// TIA Portal V19 export
VAR_GLOBAL   // PLC tag table "01_SAFETY_Q"
   FDo_C_CambioFormato_Bordatrice AT %Q1000.1 : Bool;   // 0DO1 - 169KA1/KA2
   FDo_C_HU_Pareggiatore_STO_CYTROPACK AT %Q1000.5 : Bool;   // 0DO5 - 280KA1/KA2
   FDo_C_HU_Aspo AT %Q1000.2 : Bool;   // 0DO2 - 206KA1/KA2 Motoe pompa C.Olio Aspi
   FDo_V_Air_A0301_A0302 AT %Q1558.0 : Bool;   // 200DO0 - 180YV1 - Valvola taglio aria A0301 (Ribaltamento) + A0302 ingresso (bordatrice)
   FDo_EStop_Coda_BloccaggioCremagliera_PistonePareggLong AT %Q1414.0 : Bool;   // 300DO0 - 284KA1/KA2
   FDo_V_Air_A0302_A0303 AT %Q1420.0 : Bool;   // 310DO0 - 182YV1 - Valvola taglio aria zona pareggiamento e preparazione pacco
   FDo_Ev_Stand_BY_HU_Pareggiatore AT %Q1420.1 : Bool;   // 310D01 - 282YV1
   FDo_EStop_Testa_BloccaggioCremagliera AT %Q1507.0 : Bool;   // 286KA1/KA2 - 350DO0
   FDo_C_HU_Area01 AT %Q1000.3 : Bool;   // 0DO3 - 220KA1/KA2 Motore pompa C.Olio Area 01
   FDo_C_HU_FinalCut AT %Q1000.4 : Bool;   // 0DO4 - 248KA1/KA2
   FDo_V_DecoilersHorizRot AT %Q1093.0 : Bool;   // 100DO0 - 206KA3/KA4
   FDo_V_Aspo_1 AT %Q1093.1 : Bool;   // 100DO1 - 206KA5/KA6 Contattore c/Feedback
   FDo_V_Aspo_2 AT %Q1093.2 : Bool;   // 100DO2 - 206KA7/KA8 Contattore c/Feedback
   FDo_V_CoilCar AT %Q1093.3 : Bool;   // 100DO3 - 222KA1/KA2
   FDo_V_Peeler AT %Q1093.4 : Bool;   // 100DO4 - 224KA1/KA2
   FDo_V_FinalCut AT %Q1093.5 : Bool;   // 100DO5 - 250KA1/KA2
   FDo_V_Air_Gen AT %Q1107.0 : Bool;   // 110DO0 - 174YV1
   FDo_V_StandBY_HU_Aspo AT %Q1107.1 : Bool;   // 110D01 - 208YV1
   FDo_V_StandBY_HU_Area01 AT %Q1107.2 : Bool;   // 110D02 - 221YV1
   FDo_V_Accumulatore_HU_Area01 AT %Q1107.3 : Bool;   // 110DO3 - 221YV2
   FDo_V_JB_Cut_Rest AT %Q1112.0 : Bool;   // 111DO0 - 226YV1
   FDo_V_JB_Cut_Work AT %Q1112.1 : Bool;   // 111DO1 - 226YV2
   FDo_V_StandBY_HU_FinalCut AT %Q1117.0 : Bool;   // 120DO0 - 249YV1
   FDo_V_Accumulatore_HU_FinalCut AT %Q1117.1 : Bool;   // 120DO1 - 249YV2
   FDo_C_CambioFormato_Profilatrice AT %Q1000.0 : Bool;   // 0DO0 - 168KA1/KA2
   Fdbk_V_DecoilersHorizRot_Ch1 AT %I104.6 : Bool;   // 209SQ1
   Fdbk_V_DecoilersHorizRot_Ch2 AT %I104.7 : Bool;   // 209SQ1
   Fdbk_V_Aspo01_Ch1 AT %I105.0 : Bool;   // 210SQ1
   Fdbk_V_Aspo01_Ch2 AT %I105.1 : Bool;   // 210SQ1
   Fdbk_V_Aspo02_Ch1 AT %I105.2 : Bool;   // 212SQ1
   Fdbk_V_Aspo02_Ch2 AT %I105.3 : Bool;   // 212SQ1
   Fbdk_V_CoilCar_Ch1 AT %I105.4 : Bool;   // 222SQ1
   Fbdk_V_CoilCar_Ch2 AT %I105.5 : Bool;   // 222SQ1
   Fbdk_V_Peeler_Ch1 AT %I105.6 : Bool;   // 224SQ1
   Fbdk_V_Peeler_Ch2 AT %I105.7 : Bool;   // 224SQ1
   Fbdk_V_JB_Cut_Ch1 AT %I106.0 : Bool;   // 226SQ1
   Fdbk_V_FinalCut_Ch1 AT %I108.6 : Bool;   // 250SQ1
   Fdbk_V_FinalCut_Ch2 AT %I108.7 : Bool;   // 250SQ1
   Fdbk_V_Air_Gen_Ch1 AT %I102.4 : Bool;   // 174SQ1
   Fdbk_V_Air_Gen_Ch2 AT %I102.3 : Bool;   // 174SQ1
   Fdbk_FDo_Bloccaggio_Valve AT %I360.1 : Bool;   // 286KA1/KA2
   Fbkk_C_Sezionatrice_FinalCut AT %I101.5 : Bool;   // 250KA1/KA2
   Fdbk_C_Peeler AT %I101.3 : Bool;   // 224KA1/KA2
   Fdbk_C_CoilCar AT %I101.2 : Bool;   // 222KA1/KA2
   "HU_B.Taglio_Motore_Controllo_Sicurezza" AT %I6.5 : Bool;   // 248KA1/KA2
   Fdbk_FDo_Bloccaggio_Pareggiatore_Valves AT %I309.5 : Bool;   // 284KA1
   FDo_V_Air_A0304 AT %Q1420.2 : Bool;   // 310DO2 - 183YV1
   FDo_EStop_Coda_BloccaggioCremagliera_PistonePareggLong_VS AT %I1414.0 : Bool;   // 300DO0 - 284KA1/KA2
   FDo_EStop_Testa_BloccaggioCremagliera_VS AT %I1507.0 : Bool;   // 286KA1/KA2 - 350DO0
   QBAD_FDo_C_CambioFormato_Bordatrice AT %I1000.1 : Bool;
   QBAD_FDo_C_CambioFormato_Profilatrice AT %I1000.0 : Bool;
   QBAD_FDo_C_HU_Aspo AT %I1000.2 : Bool;
   QBAD_FDo_C_HU_Area01 AT %I1000.3 : Bool;
   QBAD_FDo_C_HU_FinalCut AT %I1000.4 : Bool;
   QBAD_FDo_FDo_C_HU_Pareggiatore_STO_CYTROPACK AT %I1000.5 : Bool;
   QBAD_FDo_V_DecoilersHorizRot AT %I1093.0 : Bool;
   QBAD_FDo_V_Aspo_1 AT %I1093.1 : Bool;
   QBAD_FDo_V_Aspo_2 AT %I1093.2 : Bool;
   QBAD_FDo_V_CoilCar AT %I1093.3 : Bool;
   QBAD_FDo_V_Peeler AT %I1093.4 : Bool;
   QBAD_FDo_V_JB_Cut_Rest AT %I1112.0 : Bool;
   QBAD_FDo_V_JB_Cut_Work AT %I1112.1 : Bool;
   Fdbk_C_Aspo01 AT %I101.0 : Bool;   // 206KA5 / KA6
   Fdbk_C_Aspo02 AT %I101.1 : Bool;   // 206KA7 / KA8
   Fdbk_C_RotazioneOrizzontaleAspi AT %I100.7 : Bool;   // 206KA3 / KA4
   Fdbk_C_HU_Aspo AT %I2.2 : Bool;   // 206KA1 / KA2 Fdbk contatrore motore pompa C.Olio Aspi
   QBAD_FDo_V_FinalCut AT %I1093.5 : Bool;
   Fdbk_C_HU_Area01 AT %I2.3 : Bool;   // 220KA1 / KA2 Fdbk contatrore motore pompa C.Olio Area01
   QBAD_FDo_V_Air_Gen AT %I1107.0 : Bool;
   Fdbk_C_CambioFormato_Profilatrice AT %I2.0 : Bool;   // 168KA1
   Fdbk_C_CambioFormato_Bordatrice AT %I2.1 : Bool;   // 169KA1
   Fdbk_C_HU_Pareggiatore_STO_CYTROPACK AT %I2.4 : Bool;   // 280KA1
   QBAD_FDo_V_Air_A0301_A0302 AT %I1558.0 : Bool;
   Fdbk_V_Air_A0301_A0302_Ch1 AT %I204.7 : Bool;   // 180SQ1
   Fdbk_V_Air_A0301_A0302_Ch2 AT %I205.0 : Bool;   // 180SQ1
   Fdbk_V_Air_A0302_A0303_Ch1 AT %I300.1 : Bool;   // 182SQ1
   Fdbk_V_Air_A0302_A0303_Ch2 AT %I300.0 : Bool;   // 182SQ1
   Fdbk_V_Air_A0304_Ch1 AT %I309.7 : Bool;   // 183SQ1
   Fdbk_V_Air_A0304_Ch2 AT %I309.6 : Bool;   // 183SQ1
   QBAD_FDo_V_Air_A0302_A0303 AT %I1420.0 : Bool;
   QBAD_FDo_V_Air_A0304 AT %I1420.2 : Bool;
   Fbdk_V_JB_Cut_Ch2 AT %I106.1 : Bool;   // 226SQ1
   HU_Area02_SafetyValve AT %Q100.1 : Bool;
   "472A2_NotUsed" AT %Q1100.0 : Bool;
END_VAR
